// TIA Portal V18 export
TYPE "UDT_Vitotronic100_Alarms"
// stored: IsFailsafeCompliant false
   STRUCT
      "00 General alarm" : Array[0..2] of Bool;
   END_STRUCT;
END_TYPE
